{attribute 'qualified_only'}
{attribute 'strict'}
TYPE ENUM_PORT_STATUS :
(
	ACTIVE := 0,
	UNLOCKED := 1,
	LOCKED := 2
);
END_TYPE

(* stored: Version 1.1.0.1, ProductVersion 3.1.4024.12
   DUT ENUM_PORT_STATUS: Id {0243ee2e-9542-41eb-bd95-e56cebb740a9} *)
